PROGRAM MAIN
VAR
END_VAR

END_PROGRAM

(* stored: Version 1.1.0.1
   POU MAIN: Id {e70dbe8f-afa7-46bb-894a-4f84dee6d760} *)
